(* IEC 61131-3 sources: Temperature-Cabinet-Control-Automation/cabinet-on-off-automation, 2 files *)

(* ---- Path1_EL2869_StartStop.st ---- *)
(* =========================================================================
   Path 1 — physical on/off over EL2869 CH15/CH16, no relays (Option C).

   This is the §15 fallback: it stops BOTH the compressor and the fan by
   becoming the front-panel Start/Stop station's own 24 V supply, instead of
   trying to change anything inside the F4S. It is independent of Route A
   (RouteA_CabinetOnOff.st) — both read the same GVL_HMI.xCabinetOnCmd, so
   they can run side by side with no conflict: Route A stops the F4S's own
   control output, Path 1 cuts power to the whole station (fan included).

   Restored 31 July 2026. An earlier edit that removed Route A's lockout
   timer (per an on-site request scoped to Route A) also deleted this
   sequencer, because it shared PLC_PRG with Route A's arbitration block.
   That left xStartPulse undriven and xStopPermit hardcoded TRUE — CH15
   would never pulse and CH16 would never drop, so remote start/stop over
   EL2869 would silently do nothing on wiring landed the same day. The
   anti-short-cycle interlock here is NOT optional the way Route A's is: this
   path drives the real latching contactor directly (README §9 step 4,
   §15.2). Keep it.

   Paste into PLC_PRG as its own section, alongside Route A's section.
   Requires the GVL_HMI additions listed at the bottom, and CH15/CH16
   mapped to xStartPulse/xStopPermit in the EL2869 I/O Mapping tab
   (Always update variables = Enabled, bus cycle task = MainTask).
   ========================================================================= *)

VAR
    tonStartPulse : TON;              (* start pulse width          *)
    tonOffLock    : TON;              (* minimum off time           *)
    xCmdPrev      : BOOL;
    xRunLatch     : BOOL;             (* our view of latch state    *)
END_VAR

VAR CONSTANT
    tPULSE   : TIME := T#1S;          (* comfortably longer than latch pickup *)
    tOFFLOCK : TIME := T#5M;          (* compressor anti-short-cycle          *)
END_VAR

(* --- minimum off-time timer: runs whenever we are not running ----------- *)
tonOffLock(IN := NOT xRunLatch, PT := tOFFLOCK);
GVL_HMI.tOffLockRemain := tOFFLOCK - tonOffLock.ET;

(* --- STOP: break the series contact immediately, no interlock ----------- *)
(* Stopping is always allowed. Only starting is ever delayed. CH16 LOW
   drops the station's own supply -- Option C's remote-stop mechanism
   (README §15.4). *)
GVL_HMI.xStopPermit := GVL_HMI.xCabinetOnCmd;

IF NOT GVL_HMI.xCabinetOnCmd THEN
    xRunLatch := FALSE;
END_IF

(* --- START: rising edge, but only once the off-lock has expired --------- *)
IF GVL_HMI.xCabinetOnCmd AND NOT xCmdPrev AND tonOffLock.Q THEN
    tonStartPulse(IN := FALSE); (* reset *)
    tonStartPulse(IN := TRUE, PT := tPULSE);
    xRunLatch := TRUE;
END_IF
xCmdPrev := GVL_HMI.xCabinetOnCmd;

tonStartPulse(IN := xRunLatch AND GVL_HMI.xCabinetOnCmd, PT := tPULSE);
GVL_HMI.xStartPulse := tonStartPulse.IN AND NOT tonStartPulse.Q;

(* =========================================================================
   GVL_HMI — add (if not already present from an earlier Route A edit):

       xStartPulse    : BOOL;   (* -> EL2869 CH15, 1s pulse, parallels green button *)
       xStopPermit    : BOOL;   (* -> EL2869 CH16, TRUE = station supply live       *)
       tOffLockRemain : TIME;   (* anti-short-cycle countdown, this path only       *)

   EL2869 I/O Mapping — map two channels (README §15.3, confirmed against
   as-built drawing 7168-DWG-100 Rev B):

     CODESYS variable      | EL2869 output | -202X3 pin | Function
     xStartPulse           | CH15          | 36         | start pulse (via diode) -> wire 102
     xStopPermit           | CH16          | 37         | station supply -> wire 100
     (0 V return)           -              | 20, 29     | -> wire 101

   Before landing any wire, confirm on the meter (README §15.10 checkpoint 1)
   that the channel physically wired to pin 36 pulses ~1s and the one on
   pin 37 is steady while running -- swapping CH15/CH16 swaps a transient
   pulse for what must be a continuous supply, and Option C depends on
   that distinction.
   ========================================================================= *)

(* ---- RouteA_CabinetOnOff.st ---- *)
(* =========================================================================
   Route A — cabinet on/off over Modbus only.

   No EL2869 channel, no interposing relay, no panel wiring. The gateway
   translates the command into the F4's documented "setpoint low limit minus
   one" OFF sentinel; this POU only decides *when* to ask.

   Paste the VAR block and body into PLC_PRG (or keep it as its own POU and
   call it from PLC_PRG). Requires the GVL additions listed at the bottom and
   two new Modbus TCP channels.

   No anti-short-cycle interlock here — removed 31 July 2026 by field
   decision so the cabinet responds instantly to xCabinetOnCmd from CODESYS.
   This trades away the compressor protection the mechanical/EL2869 path
   (Path1_EL2869_StartStop.st) still keeps; Test 3 in that day's field
   session rapid-cycled the real compressor five times with no minimum
   off-time to confirm the change took effect. If Route A ever becomes the
   only path commanding the compressor (i.e. Path 1 is not also wired), put
   a minimum off-time back before relying on this for daily use.
   ========================================================================= *)

(* --- Command arbitration ------------------------------------------------ *)
(* STOP is immediate and unconditional. START is immediate too — no lockout,
   no gate. See the header note above for the trade-off this makes. *)
IF NOT GVL_HMI.xCabinetOnCmd THEN
    GVL_Modbus.wOnOffCmd := 1;                    (* 1 = OFF *)
ELSE
    GVL_Modbus.wOnOffCmd := 2;                    (* 2 = ON *)
END_IF

(* --- Feedback ----------------------------------------------------------- *)
(* wOnOffState is derived by the gateway from F4 register 300 as read back,
   not from the last command, so this is observation and not an echo. It is
   still only proof that the *controller output* is enabled — see README
   section 16 on what it does and does not prove about the fan. *)
GVL_HMI.xCabinetRunning := (GVL_Modbus.wOnOffState = 2);

(* xStopPermit is NOT written here. It belongs to
   Path1_EL2869_StartStop.st, which drives EL2869 CH16 from it. If both
   sections write it, whichever runs later in the scan wins every cycle —
   if that happened to be this one, CH16 would be forced permanently HIGH
   and Path 1's remote stop would silently stop working. If Path 1 is not
   pasted into this PLC_PRG, xStopPermit is simply unused; do not "fix"
   that by writing TRUE here again. *)

(* =========================================================================
   GVL_Modbus — add:

       wOnOffCmd     : WORD;   (* 0 = none, 1 = off, 2 = on   -> gateway *)
       wOnOffState   : WORD;   (* 0 = unknown, 1 = off, 2 = on <- gateway *)
       wSpLowLimit   : WORD;   (* F4 setpoint low limit, signed x10        *)
       wProfileNow   : WORD;   (* running profile number, 0 = none         *)

   GVL_HMI — xStartPulse and xStopPermit are NOT Route A's. They belong to
   Path1_EL2869_StartStop.st (EL2869 CH15/CH16, README §15). Route A only
   ever touches wOnOffCmd, xCabinetRunning and xCabinetOnCmd (input). Do not
   add writes to xStartPulse/xStopPermit here even if both POUs are pasted
   into the same PLC_PRG — see the comment at the feedback block above.

   Modbus TCP Slave channels to add (element row, type WORD, as with every
   existing channel in this project):

     # | Access                        | Trigger        | Offset  | Maps to
     5 | Write Single Register (FC06)  | Cyclic 1000 ms | 16#0005 | wOnOffCmd
     6 | Read Holding Registers (FC03) | Cyclic 1000 ms | 16#0006 | wOnOffState
     7 | Read Holding Registers (FC03) | Cyclic 1000 ms | 16#0007 | wSpLowLimit
     8 | Read Holding Registers (FC03) | Cyclic 1000 ms | 16#0008 | wProfileNow

   Channels 7 and 8 are diagnostics — the OFF sentinel the gateway derived,
   and whether a profile is running. Neither is required for on/off to work.

   Bus cycle task must be MainTask and "Always update variables" enabled,
   the same setting that channels 0-4 needed.
   ========================================================================= *)
